// Mitsubishi GX Works2 project: servo3   PLC: Q03UDV

PROGRAM MAIN
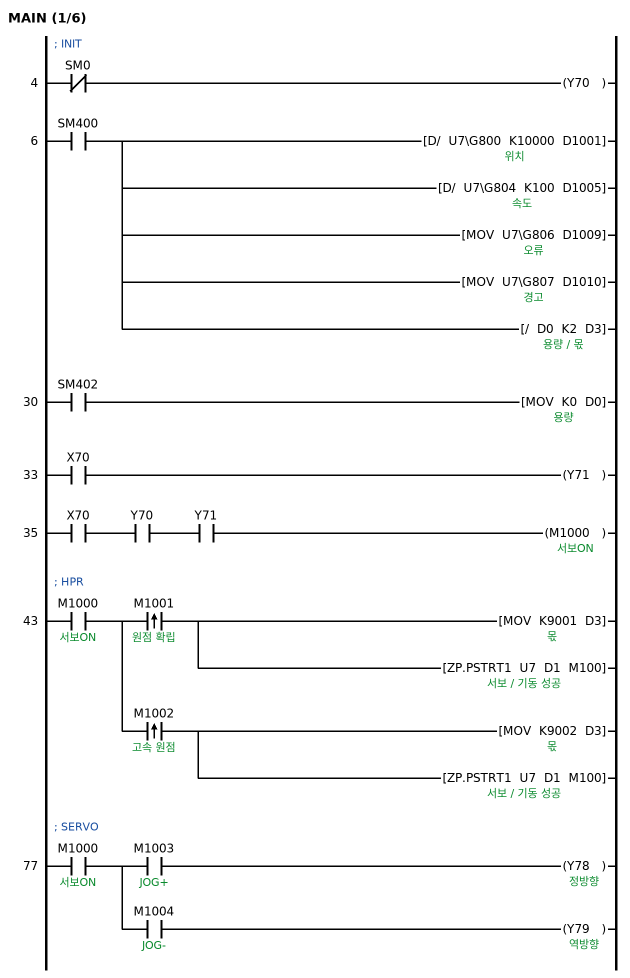
; INIT
4     LDI     SM0
      OUT     Y70
6     LD      SM400
      D/      U7\G800 K10000 D1001  ; 위치
      D/      U7\G804 K100 D1005  ; 속도
      MOV     U7\G806 D1009  ; 오류
      MOV     U7\G807 D1010  ; 경고
      /       D0 K2 D3  ; 용량 / 몫
30    LD      SM402
      MOV     K0 D0
33    LD      X70
      OUT     Y71
35    LD      X70
      AND     Y70
      AND     Y71
      OUT     M1000  ; 서보ON
; HPR
43    LD      M1000  ; 서보ON
      MPS
      ANDP    M1001  ; 원점 확립
      MOV     K9001 D3
      ZP.PSTRT1 U7 D1 M100  ; 서보 / 기동 성공
      MPP
      ANDP    M1002  ; 고속 원점
      MOV     K9002 D3
      ZP.PSTRT1 U7 D1 M100
; SERVO
77    LD      M1000  ; 서보ON
      MPS
      AND     M1003  ; JOG+
      OUT     Y78  ; 정방향
      MPP
      AND     M1004  ; JOG-
      OUT     Y79  ; 역방향
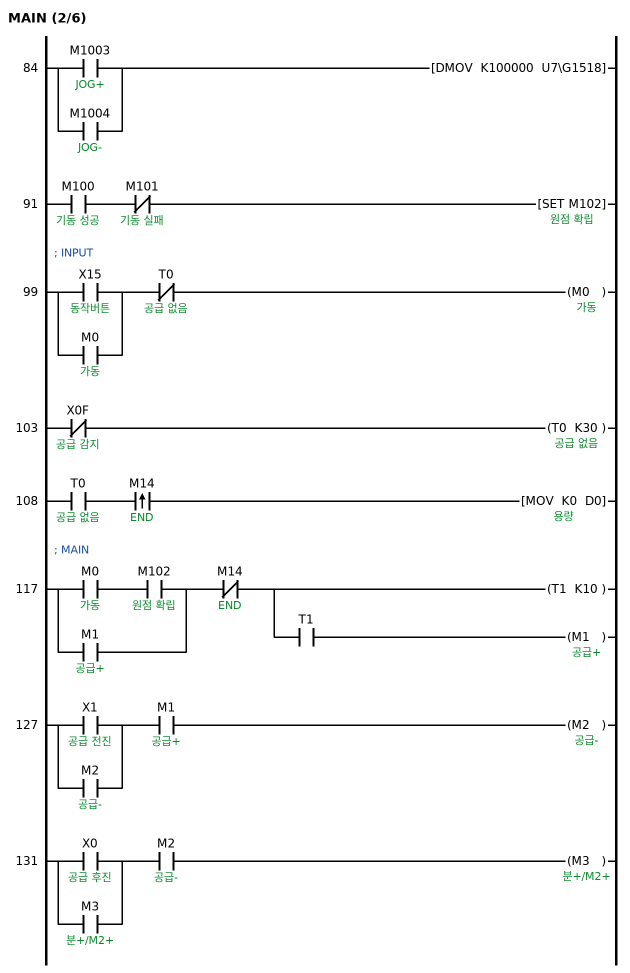
84    LD      M1003  ; JOG+
      OR      M1004  ; JOG-
      DMOV    K100000 U7\G1518
91    LD      M100  ; 기동 성공
      ANI     M101  ; 기동 실패
      SET     M102  ; 원점 확립
; INPUT
99    LD      X15  ; 동작버튼
      OR      M0  ; 가동
      ANI     T0  ; 공급 없음
      OUT     M0  ; 가동
103   LDI     X0F  ; 공급 감지
      OUT     T0 K30  ; 공급 없음
108   LD      T0  ; 공급 없음
      ANDP    M14  ; END
      MOV     K0 D0
; MAIN
117   LD      M0  ; 가동
      AND     M102  ; 원점 확립
      OR      M1  ; 공급+
      ANI     M14  ; END
      OUT     T1 K10
      AND     T1
      OUT     M1  ; 공급+
127   LD      X1  ; 공급 전진
      OR      M2  ; 공급-
      AND     M1  ; 공급+
      OUT     M2  ; 공급-
131   LD      X0  ; 공급 후진
      OR      M3  ; 분+/M2+
      AND     M2  ; 공급-
      OUT     M3  ; 분+/M2+
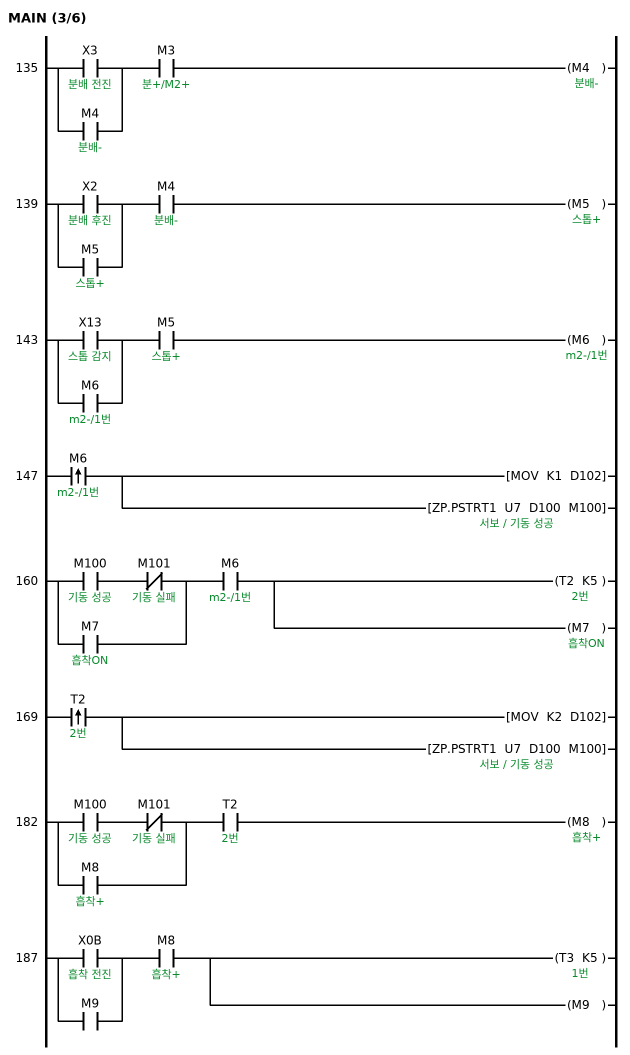
135   LD      X3  ; 분배 전진
      OR      M4  ; 분배-
      AND     M3  ; 분+/M2+
      OUT     M4  ; 분배-
139   LD      X2  ; 분배 후진
      OR      M5  ; 스톱+
      AND     M4  ; 분배-
      OUT     M5  ; 스톱+
143   LD      X13  ; 스톱 감지
      OR      M6  ; m2-/1번
      AND     M5  ; 스톱+
      OUT     M6  ; m2-/1번
147   LDP     M6  ; m2-/1번
      MOV     K1 D102
      ZP.PSTRT1 U7 D100 M100
160   LD      M100  ; 기동 성공
      ANI     M101  ; 기동 실패
      OR      M7  ; 흡착ON
      AND     M6  ; m2-/1번
      OUT     T2 K5  ; 2번
      OUT     M7  ; 흡착ON
169   LDP     T2  ; 2번
      MOV     K2 D102
      ZP.PSTRT1 U7 D100 M100
182   LD      M100  ; 기동 성공
      ANI     M101  ; 기동 실패
      OR      M8  ; 흡착+
      AND     T2  ; 2번
      OUT     M8  ; 흡착+
187   LD      X0B  ; 흡착 전진
      OR      M9
      AND     M8  ; 흡착+
      OUT     T3 K5  ; 1번
      OUT     M9
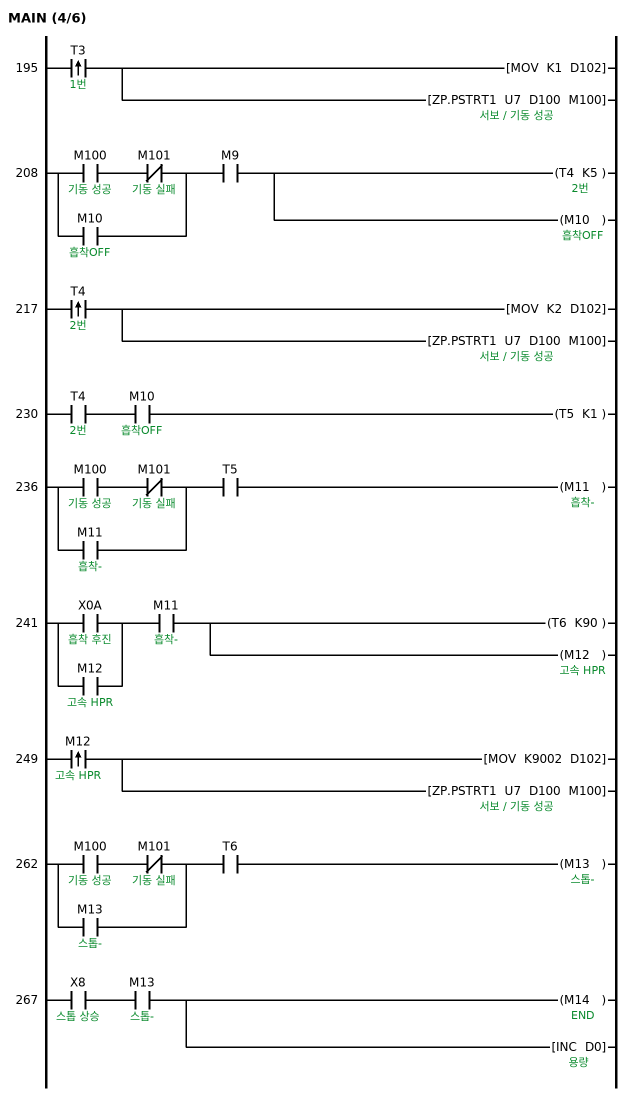
195   LDP     T3  ; 1번
      MOV     K1 D102
      ZP.PSTRT1 U7 D100 M100
208   LD      M100  ; 기동 성공
      ANI     M101  ; 기동 실패
      OR      M10  ; 흡착OFF
      AND     M9
      OUT     T4 K5  ; 2번
      OUT     M10  ; 흡착OFF
217   LDP     T4  ; 2번
      MOV     K2 D102
      ZP.PSTRT1 U7 D100 M100
230   LD      T4  ; 2번
      AND     M10  ; 흡착OFF
      OUT     T5 K1
236   LD      M100  ; 기동 성공
      ANI     M101  ; 기동 실패
      OR      M11  ; 흡착-
      AND     T5
      OUT     M11  ; 흡착-
241   LD      X0A  ; 흡착 후진
      OR      M12  ; 고속 HPR
      AND     M11  ; 흡착-
      OUT     T6 K90
      OUT     M12  ; 고속 HPR
249   LDP     M12  ; 고속 HPR
      MOV     K9002 D102
      ZP.PSTRT1 U7 D100 M100
262   LD      M100  ; 기동 성공
      ANI     M101  ; 기동 실패
      OR      M13  ; 스톱-
      AND     T6
      OUT     M13  ; 스톱-
267   LD      X8  ; 스톱 상승
      AND     M13  ; 스톱-
      OUT     M14  ; END
      INC     D0
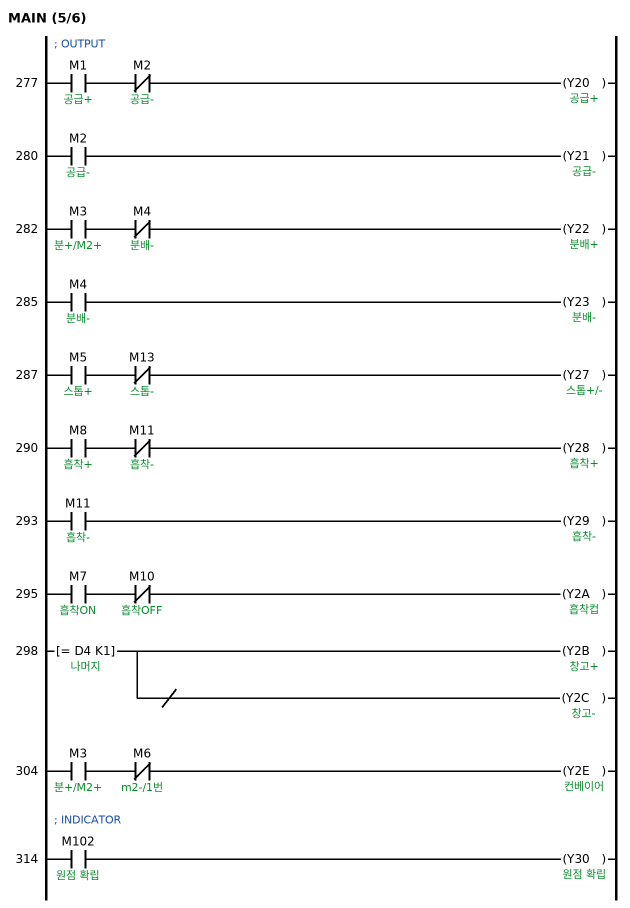
; OUTPUT
277   LD      M1  ; 공급+
      ANI     M2  ; 공급-
      OUT     Y20  ; 공급+
280   LD      M2  ; 공급-
      OUT     Y21  ; 공급-
282   LD      M3  ; 분+/M2+
      ANI     M4  ; 분배-
      OUT     Y22  ; 분배+
285   LD      M4  ; 분배-
      OUT     Y23  ; 분배-
287   LD      M5  ; 스톱+
      ANI     M13  ; 스톱-
      OUT     Y27  ; 스톱+/-
290   LD      M8  ; 흡착+
      ANI     M11  ; 흡착-
      OUT     Y28  ; 흡착+
293   LD      M11  ; 흡착-
      OUT     Y29  ; 흡착-
295   LD      M7  ; 흡착ON
      ANI     M10  ; 흡착OFF
      OUT     Y2A  ; 흡착컵
298   LD=     D4 K1  ; 나머지
      OUT     Y2B  ; 창고+
      INV
      OUT     Y2C  ; 창고-
304   LD      M3  ; 분+/M2+
      ANI     M6  ; m2-/1번
      OUT     Y2E  ; 컨베이어
; INDICATOR
314   LD      M102  ; 원점 확립
      OUT     Y30  ; 원점 확립
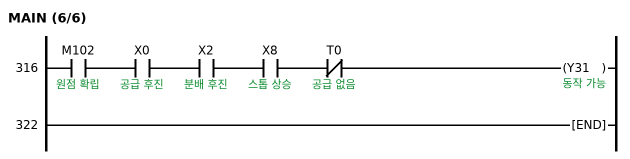
316   LD      M102  ; 원점 확립
      AND     X0  ; 공급 후진
      AND     X2  ; 분배 후진
      AND     X8  ; 스톱 상승
      ANI     T0  ; 공급 없음
      OUT     Y31  ; 동작 가능
322   END
END_PROGRAM

// device comments not shown above
X9  ; 스톱 하강
D2  ; 몫
M1005  ; 에러 리셋
